(* PLC project CodesysTest.project, PN2IC PLCopen CODESYS V3.5 SP17 Patch 3 *)
(* stored: creationDateTime 2022-12-11T22:12:36, modificationDateTime 2022-12-11T22:12:36 *)

PROGRAM flow_1

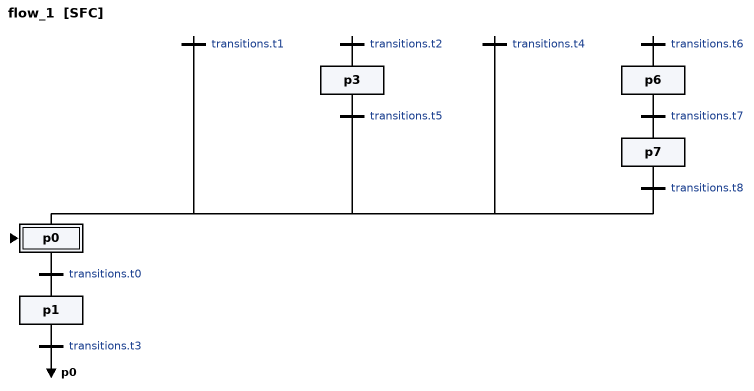
INITIAL_STEP p0:
END_STEP
TRANSITION FROM p0 TO p1
  := transitions.t0;
END_TRANSITION
STEP p1:
END_STEP
TRANSITION FROM p1 TO p0
  := transitions.t3;
END_TRANSITION
STEP p3:
END_STEP
TRANSITION FROM p3 TO p0
  := transitions.t5;
END_TRANSITION
STEP p6:
END_STEP
TRANSITION FROM p6 TO p7
  := transitions.t7;
END_TRANSITION
STEP p7:
END_STEP
TRANSITION FROM p7 TO p0
  := transitions.t8;
END_TRANSITION
TRANSITION FROM ? TO p0
  := transitions.t1;
END_TRANSITION
TRANSITION FROM ? TO p3
  := transitions.t2;
END_TRANSITION
TRANSITION FROM ? TO p0
  := transitions.t4;
END_TRANSITION
TRANSITION FROM ? TO p6
  := transitions.t6;
END_TRANSITION
END_PROGRAM

PROGRAM transitions

         
        
END_PROGRAM

CONFIGURATION Application
  RESOURCE Application ON PLC
    VAR_GLOBAL  (* GVL *)
      t5 : BOOL;
      t1 : BOOL;
      t6 : BOOL;
      t0 : BOOL;
      t7 : BOOL;
      t2 : BOOL;
      t8 : BOOL;
      t4 : BOOL;
      t3 : BOOL;
    END_VAR
    TASK MainTask(INTERVAL := T#20ms, PRIORITY := 1);
    PROGRAM flow_1 WITH MainTask : flow_1;
  END_RESOURCE
END_CONFIGURATION
